// TwinCAT 3 PLC project Practice_1
// ProgramVersion: 3.1.4024.0
// libraries:
//   Tc2_Standard, * (Beckhoff Automation GmbH)
//   Tc2_System, * (Beckhoff Automation GmbH)
//   Tc3_Module, * (Beckhoff Automation GmbH)
// project tree:
//   GVLs/ GVL.TcGVL
//   / PlcTask.TcTTO
//   POUs/ MAIN.TcPOU
// real-time tasks:
//   TASK PlcTask: cycle T#10ms, priority 20, ADS port 350
//   TASK PlcTask1: cycle T#10ms, priority 21, ADS port 351
//   TASK PlcTask2: cycle T#10ms, priority 22, ADS port 352

CONFIGURATION Practice_1
    RESOURCE PLC ON TwinCAT3
        TASK PlcTask(INTERVAL := T#10ms, PRIORITY := 20);
        PROGRAM MAIN WITH PlcTask : MAIN;
    END_RESOURCE
END_CONFIGURATION

// ---- GVLs/GVL.TcGVL
{attribute 'qualified_only'}
VAR_GLOBAL
	bStart : BOOL;
	nCount : INT ;
END_VAR

// ---- POUs/MAIN.TcPOU
PROGRAM MAIN
VAR
	bRunning : BOOL;
END_VAR

IF GVL.bStart THEN
	GVL.nCount := GVL.nCount + 1;
	//GVL.bStart := FALSE;
	bRunning := TRUE;
ELSE
	bRunning := FALSE;
END_IF

END_PROGRAM
